FUNCTION_BLOCK GUYSON_AI_CTRL
VAR_INPUT

	BOOL_ST :BOOL; (*Analog Data Collection Start Bit*)
	INT_M1_AI :INT; (*Guyson Generator Master 1 Analog Input Data*)
	INT_M2_AI :INT; (*Guyson Generator Master 2 Analog Input Data*)
	TIME_REFRESH :TIME; (*Refresh Time assigned*)
	TIME_DATA_COLLECT :TIME; (*Delay time for data collection for stability improvement, This data must be ALWAYS "Half" or below from "TIME_REFRESH" SetPoint *)

END_VAR

VAR_OUTPUT

	M1CH1_INT :INT; (*ANALOG READING OF MASTER1-CHANNEL1*)
	M1CH2_INT :INT; (*ANALOG READING OF MASTER1-CHANNEL2*)
	S1CH1_INT :INT; (*ANALOG READING OF SLAVE1-CHANNEL1*)
	M2CH1_INT :INT; (*ANALOG READING OF MASTER2-CHANNEL1*)
	M2CH2_INT :INT; (*ANALOG READING OF MASTER2-CHANNEL2*)
	S2CH1_INT :INT; (*ANALOG READING OF SLAVE2-CHANNEL1*)
	M1_PIN1_DO_BOOL :BOOL; (*GUYSON MASTER 1 SCADA CONNECTOR PIN 1 (A0) CONNECTION OUTPUT FOR MODULE SELECTION*)
	M1_PIN7_DO_BOOL :BOOL; (*GUYSON MASTER 1 SCADA CONNECTOR PIN 7 (A3) CONNECTION OUTPUT FOR IDENTITY SELECTION*)
	M2_PIN1_DO_BOOL :BOOL; (*GUYSON MASTER 2 SCADA CONNECTOR PIN 1 (A0) CONNECTION OUTPUT FOR MODULE SELECTION*)
	M2_PIN7_DO_BOOL :BOOL; (*GUYSON MASTER 2 SCADA CONNECTOR PIN 7 (A3) CONNECTION OUTPUT FOR IDENTITY SELECTION*)
	IT1AOUT_BOOL: BOOL;
	IT2AOUT_BOOL: BOOL;
	IT3AOUT_BOOL: BOOL;
	IT1BOUT_BOOL: BOOL;
	IT2BOUT_BOOL: BOOL;
	IT3BOUT_BOOL: BOOL;





END_VAR
VAR
	IT1A: TON;
	IT2A: TON;
	IT3A: TON;
	IT1B: TON;
	IT2B: TON;
	IT3B: TON;


	M1CH1BOOLOUT: BOOL;
	M1CH2BOOLOUT: BOOL;
	S1CH1BOOLOUT: BOOL;
	M2CH1BOOLOUT: BOOL;
	M2CH2BOOLOUT: BOOL;
	S2CH1BOOLOUT: BOOL;

END_VAR
VAR // added by the converter: edge detectors and wires of the graphical bodies
    _w1, _w2, _w3 : BOOL;
    _w4, _w5, _w6, _w7, _w8, _w9 : INT;
END_VAR

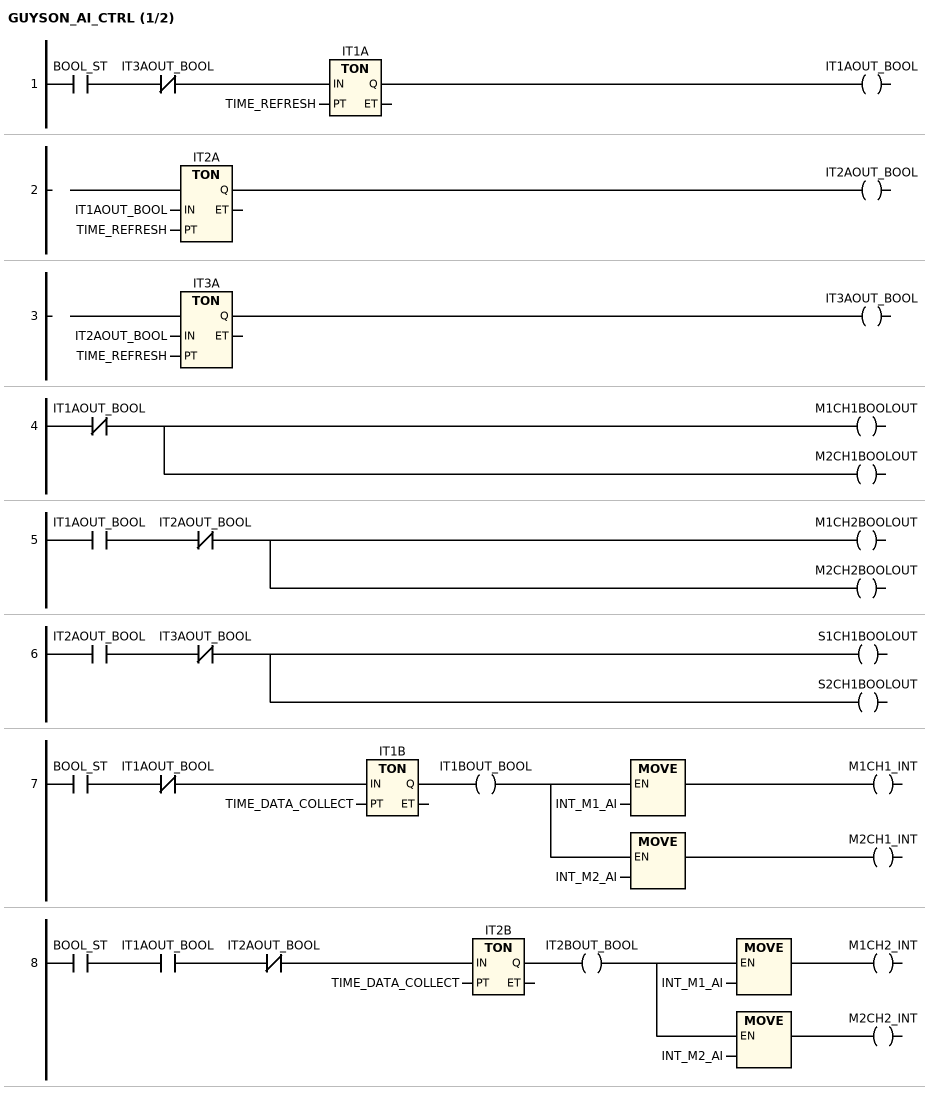
// NETWORK 1
IT1A(IN := BOOL_ST AND NOT IT3AOUT_BOOL, PT := TIME_REFRESH); // TON
IT1AOUT_BOOL := IT1A.Q;

// NETWORK 2
IT2A(IN := IT1AOUT_BOOL, PT := TIME_REFRESH); // TON
IT2AOUT_BOOL := IT2A.Q;

// NETWORK 3
IT3A(IN := IT2AOUT_BOOL, PT := TIME_REFRESH); // TON
IT3AOUT_BOOL := IT3A.Q;

// NETWORK 4
_w1 := NOT IT1AOUT_BOOL;
M1CH1BOOLOUT := _w1;
M2CH1BOOLOUT := _w1;

// NETWORK 5
_w2 := IT1AOUT_BOOL AND NOT IT2AOUT_BOOL;
M1CH2BOOLOUT := _w2;
M2CH2BOOLOUT := _w2;

// NETWORK 6
_w3 := IT2AOUT_BOOL AND NOT IT3AOUT_BOOL;
S1CH1BOOLOUT := _w3;
S2CH1BOOLOUT := _w3;

// NETWORK 7
IT1B(IN := BOOL_ST AND NOT IT1AOUT_BOOL, PT := TIME_DATA_COLLECT); // TON
IT1BOUT_BOOL := IT1B.Q;
IF IT1B.Q THEN _w4 := INT_M1_AI; END_IF
M1CH1_INT := _w4;
IF IT1B.Q THEN _w5 := INT_M2_AI; END_IF
M2CH1_INT := _w5;

// NETWORK 8
IT2B(IN := BOOL_ST AND IT1AOUT_BOOL AND NOT IT2AOUT_BOOL, PT := TIME_DATA_COLLECT); // TON
IT2BOUT_BOOL := IT2B.Q;
IF IT2B.Q THEN _w6 := INT_M1_AI; END_IF
M1CH2_INT := _w6;
IF IT2B.Q THEN _w7 := INT_M2_AI; END_IF
M2CH2_INT := _w7;

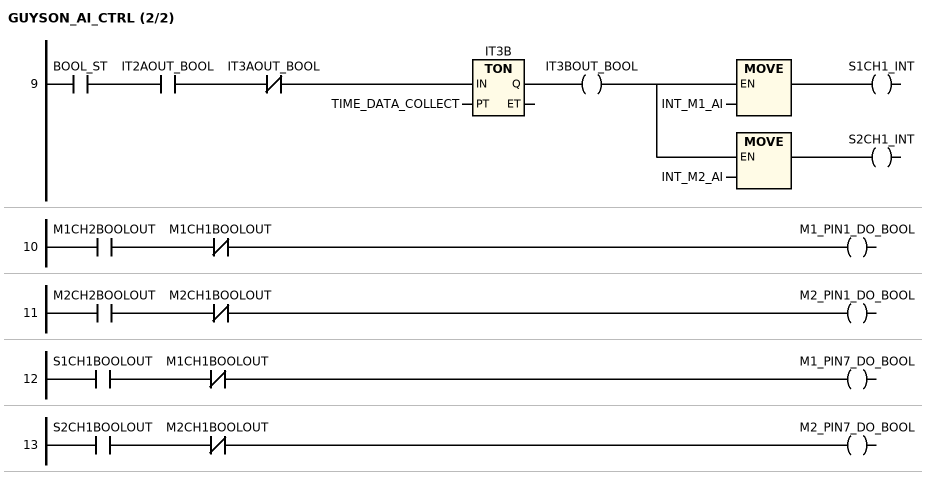
// NETWORK 9
IT3B(IN := BOOL_ST AND IT2AOUT_BOOL AND NOT IT3AOUT_BOOL, PT := TIME_DATA_COLLECT); // TON
IT3BOUT_BOOL := IT3B.Q;
IF IT3B.Q THEN _w8 := INT_M1_AI; END_IF
S1CH1_INT := _w8;
IF IT3B.Q THEN _w9 := INT_M2_AI; END_IF
S2CH1_INT := _w9;

// NETWORK 10
M1_PIN1_DO_BOOL := M1CH2BOOLOUT AND NOT M1CH1BOOLOUT;

// NETWORK 11
M2_PIN1_DO_BOOL := M2CH2BOOLOUT AND NOT M2CH1BOOLOUT;

// NETWORK 12
M1_PIN7_DO_BOOL := S1CH1BOOLOUT AND NOT M1CH1BOOLOUT;

// NETWORK 13
M2_PIN7_DO_BOOL := S2CH1BOOLOUT AND NOT M2CH1BOOLOUT;

END_FUNCTION_BLOCK

(* stored: Version 1.1.0.1, ProductVersion 3.1.4024.12
   POU GUYSON_AI_CTRL: Id {5773d6a7-eed3-4419-ac21-f6fe0e92cf41}, SpecialFunc None *)
